PROGRAM fileio3
VAR
	bdo:BOOL;
	rdo:R_trig;

	fopen:FB_FileOPen;
	fclose:FB_Fileclose;
	fRead:FB_FileRead;
	fGet:FB_FileGets;
	state: INT := 0;
	buffRead                        :ARRAY[1..1000] OF BYTE;
	cbcount : UDINT;
	outstr : string;
END_VAR

rdo(clk := bdo);

CASE state OF
	0:
		IF rdo.Q THEN
			bdo:=FALSE;
			state :=1;
		END_IF
	1:
			fopen(
				sPathName := 'C:\0 0json\scan.json',
				nMode := FOPEN_MODEREAD OR FOPEN_MODETEXT,
				bExecute := TRUE,
				tTimeout := T#15S);
				
				IF fopen.bBusy AND NOT fopen.bError THEN
					state := 2;
				END_IF
	2: 
			fRead(
				hFile:=fopen.hFile,
				pReadBuff:= ADR(buffRead), 
				cbReadLen:= SIZEOF(buffRead),
				cbRead => cbcount,
				bExecute:=TRUE, 
				tTimeout:=T#15S);

				IF fRead.bBusy AND NOT fRead.bError THEN
					state := 3;
				END_IF
	4: 
			fget(hfile:=fopen.hFile, bExecute := TRUE, TTimeout := T#15S);
			outstr := fget.sLine;
			
				IF fget.bBusy AND NOT fget.bError THEN
					state := 3;
				END_IF
	3:
		fclose(hFile := fopen.hFile,
				bExecute := TRUE,
				tTimeout:=T#5S);
			IF fclose.bBusy AND NOT fclose.bError THEN
				state := 0;
			END_IF
			
	ELSE
		state := 0;
END_CASE

END_PROGRAM

(* stored: Version 1.1.0.1, ProductVersion 3.1.4024.2
   POU fileio3: Id {654dd14c-9787-456c-af97-d53e4a191c15}, SpecialFunc None *)
